PROGRAM P_System
VAR
END_VAR

P_FootPedal();
P_SystemEnvironment();
P_SafetyGuard();

END_PROGRAM

(* stored: Version 1.1.0.1, ProductVersion 3.1.4024.11
   POU P_System: Id {c09b011e-c062-4ba7-b851-1efa888f388a}, SpecialFunc None *)
